TYPE SwitchInfo :
STRUCT
	
END_STRUCT
END_TYPE

(* stored: Version 1.1.0.1, ProductVersion 3.1.4024.11
   DUT SwitchInfo: Id {7c92b0d9-0eb1-40a5-894d-4ea93633db70} *)
